{attribute 'qualified_only'}
VAR_GLOBAL
	//Shaft Ramp Supply
	PSU1_OK				: BOOL := FALSE;
	VMB 				: ST_VoltMon_Base;
	SegmentCharged		: BOOL := FALSE;
	CloseSRChargeRly	: BOOL := FALSE;
	SRChargeRly_close 	: BOOL := FALSE;
	OpenSRDumpRly		: ARRAY[1..8] OF BOOL;
	SRDumpRelay_close 	: BOOL := FALSE;
END_VAR

(* stored: Version 1.1.0.1, ProductVersion 3.1.4024.11
   GVL LCP3_IO: Id {1740c835-4b09-49d2-9d11-138c7e138ab6} *)
